FUNCTION_BLOCK AW_TO_AL (* Composite FB for converting AW (WORD) adapter to AL (LWORD) adapter *)
  (* Standard: 61499-2; Description: Copyright (c) 2026 HR Agrartechnik GmbH This program and the accompanying materials are made available under the terms of the Eclipse Public License 2.0 which is available at https://www.eclipse.org/legal/epl-2.0/ SPDX-License-Identifier: EPL-2.0 *)
  (* Version 1.0, 2026-02-17, Franz Höpfinger, HR Agrartechnik GmbH *)
  PACKAGE adapter::conversion::unidirectional;
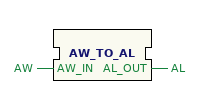
  SOCKETS
    AW_IN : adapter::types::unidirectional::AW; (* WORD Adapter Input *)
  END_SOCKETS
  PLUGS
    AL_OUT : adapter::types::unidirectional::AL; (* LWORD Adapter Output *)
  END_PLUGS
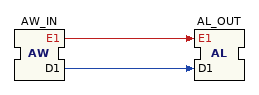
  EVENT_CONNECTIONS
    AW_IN.E1 TO AL_OUT.E1;
  END_CONNECTIONS
  DATA_CONNECTIONS
    AW_IN.D1 TO AL_OUT.D1;
  END_CONNECTIONS
END_FUNCTION_BLOCK
